{attribute 'qualified_only'}
VAR_GLOBAL
    // =====================================================
    // TwinCAT NC轴引用
    // 当前只声明一根测试轴
    // 建立NC轴后，将PlcToNc和NcToPlc与NC轴链接
    // =====================================================
    Axis1Ref : AXIS_REF;			// TwinCAT NC轴引用
END_VAR

(* stored: Version 1.1.0.1, ProductVersion 3.1.4026.18
   GVL GVL_AxisRef: Id {3b459897-13ae-4f42-9e85-8d77d1facf15} *)
